{attribute addProperty BoxType "IODEVICETYPE_ETHERCATPROT"}
{attribute addProperty Id "WcStateAT %I*BIT10.1250"}
{attribute addProperty CRC "682125173"}
{attribute addProperty SizeInBites "1"}
{attribute addProperty SizeInBytes "0.125"}
TYPE WcState_28A86775 :
STRUCT
	{attribute addProperty Name "WcState"}
	WcState AT %I* : BIT;
END_STRUCT
END_TYPE

(* stored: Version 1.2.0.0, ProductVersion 3.1.4024.9
   DUT WcState_28A86775: Id {b55ab08b-3f56-42e0-bc04-24d44711f059} *)
